// Mitsubishi GX Works2 project: 23_5   PLC: Q03UDV

PROGRAM MAIN
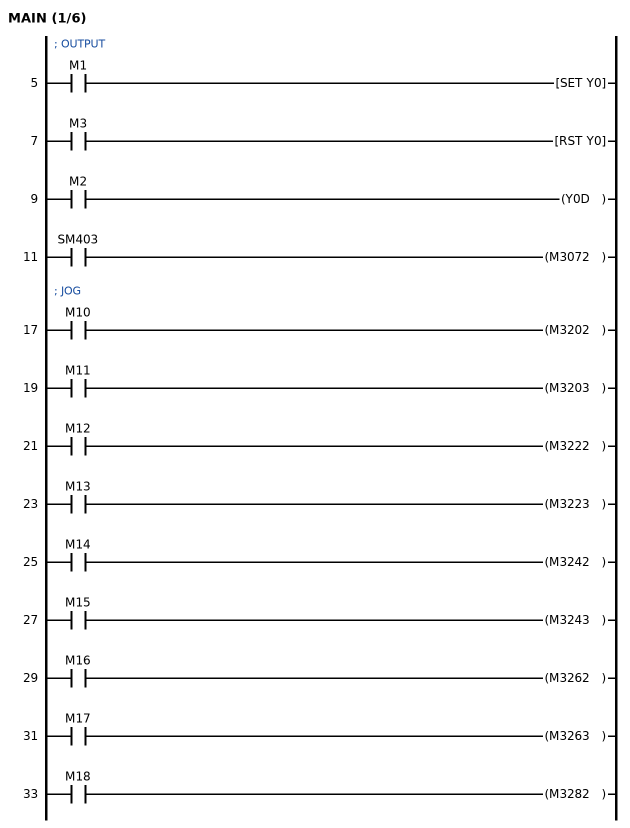
; OUTPUT
5     LD      M1
      SET     Y0
7     LD      M3
      RST     Y0
9     LD      M2
      OUT     Y0D
11    LD      SM403
      OUT     M3072
; JOG
17    LD      M10
      OUT     M3202
19    LD      M11
      OUT     M3203
21    LD      M12
      OUT     M3222
23    LD      M13
      OUT     M3223
25    LD      M14
      OUT     M3242
27    LD      M15
      OUT     M3243
29    LD      M16
      OUT     M3262
31    LD      M17
      OUT     M3263
33    LD      M18
      OUT     M3282
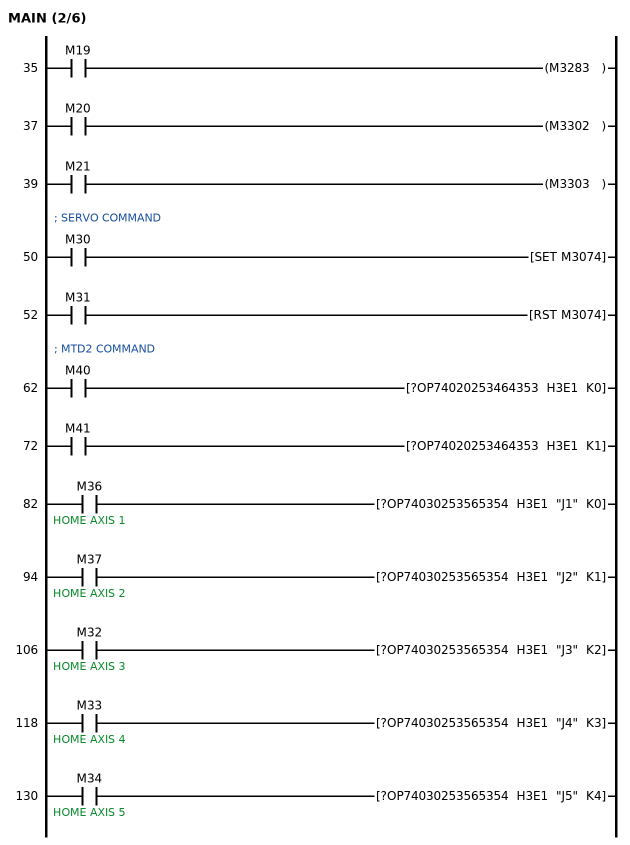
35    LD      M19
      OUT     M3283
37    LD      M20
      OUT     M3302
39    LD      M21
      OUT     M3303
; SERVO COMMAND
50    LD      M30
      SET     M3074
52    LD      M31
      RST     M3074
; MTD2 COMMAND
62    LD      M40
      ?OP74020253464353 H3E1 K0
72    LD      M41
      ?OP74020253464353 H3E1 K1
82    LD      M36  ; HOME AXIS 1
      ?OP74030253565354 H3E1 "J1" K0
94    LD      M37  ; HOME AXIS 2
      ?OP74030253565354 H3E1 "J2" K1
106   LD      M32  ; HOME AXIS 3
      ?OP74030253565354 H3E1 "J3" K2
118   LD      M33  ; HOME AXIS 4
      ?OP74030253565354 H3E1 "J4" K3
130   LD      M34  ; HOME AXIS 5
      ?OP74030253565354 H3E1 "J5" K4
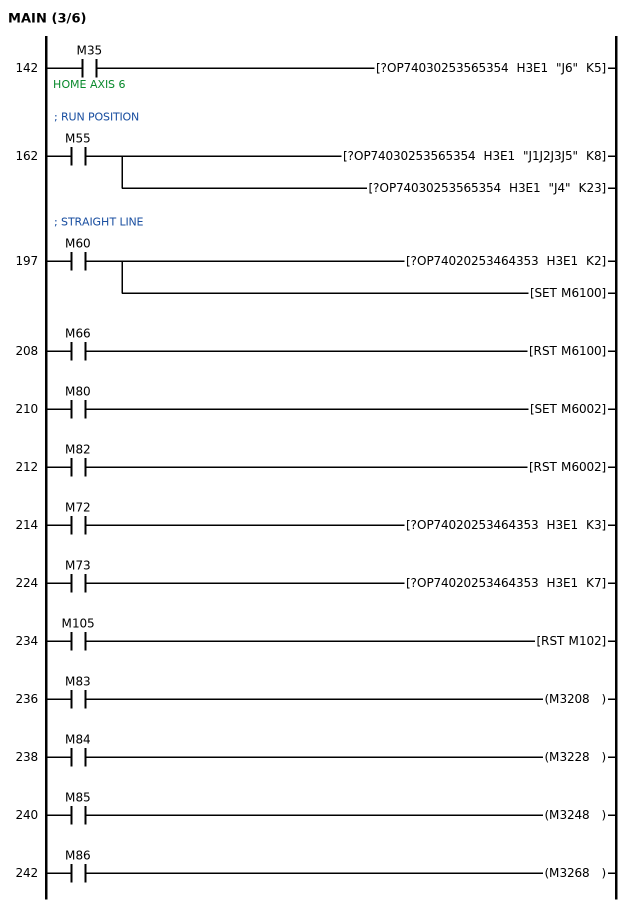
142   LD      M35  ; HOME AXIS 6
      ?OP74030253565354 H3E1 "J6" K5
; RUN POSITION
162   LD      M55
      ?OP74030253565354 H3E1 "J1J2J3J5" K8
      ?OP74030253565354 H3E1 "J4" K23
; STRAIGHT LINE
197   LD      M60
      ?OP74020253464353 H3E1 K2
      SET     M6100
208   LD      M66
      RST     M6100
210   LD      M80
      SET     M6002
212   LD      M82
      RST     M6002
214   LD      M72
      ?OP74020253464353 H3E1 K3
224   LD      M73
      ?OP74020253464353 H3E1 K7
234   LD      M105
      RST     M102
236   LD      M83
      OUT     M3208
238   LD      M84
      OUT     M3228
240   LD      M85
      OUT     M3248
242   LD      M86
      OUT     M3268
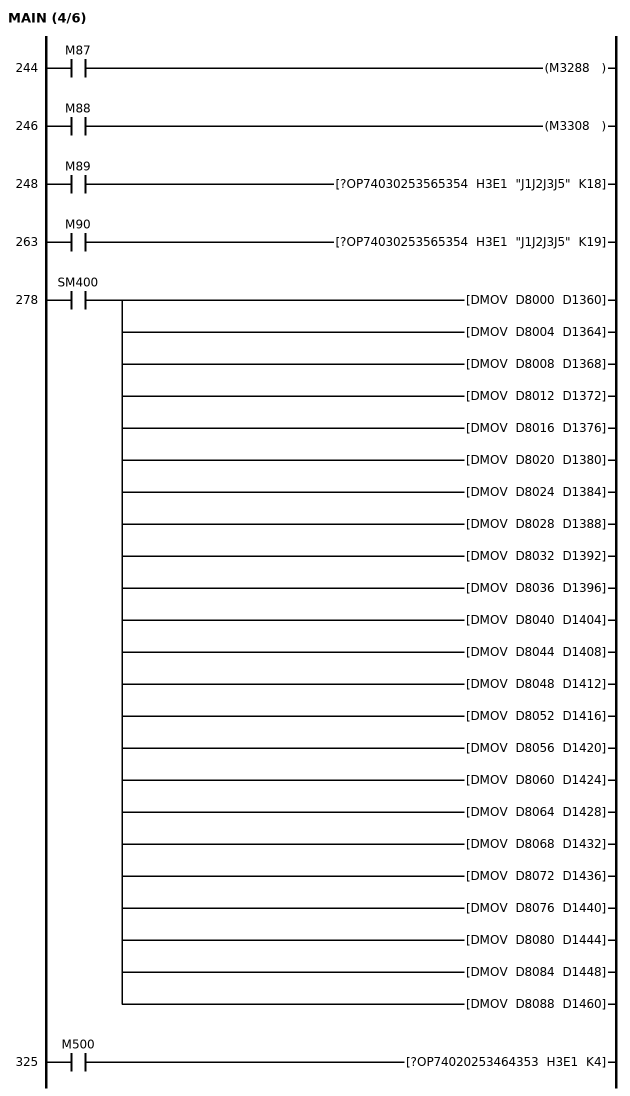
244   LD      M87
      OUT     M3288
246   LD      M88
      OUT     M3308
248   LD      M89
      ?OP74030253565354 H3E1 "J1J2J3J5" K18
263   LD      M90
      ?OP74030253565354 H3E1 "J1J2J3J5" K19
278   LD      SM400
      DMOV    D8000 D1360
      DMOV    D8004 D1364
      DMOV    D8008 D1368
      DMOV    D8012 D1372
      DMOV    D8016 D1376
      DMOV    D8020 D1380
      DMOV    D8024 D1384
      DMOV    D8028 D1388
      DMOV    D8032 D1392
      DMOV    D8036 D1396
      DMOV    D8040 D1404
      DMOV    D8044 D1408
      DMOV    D8048 D1412
      DMOV    D8052 D1416
      DMOV    D8056 D1420
      DMOV    D8060 D1424
      DMOV    D8064 D1428
      DMOV    D8068 D1432
      DMOV    D8072 D1436
      DMOV    D8076 D1440
      DMOV    D8080 D1444
      DMOV    D8084 D1448
      DMOV    D8088 D1460
325   LD      M500
      ?OP74020253464353 H3E1 K4
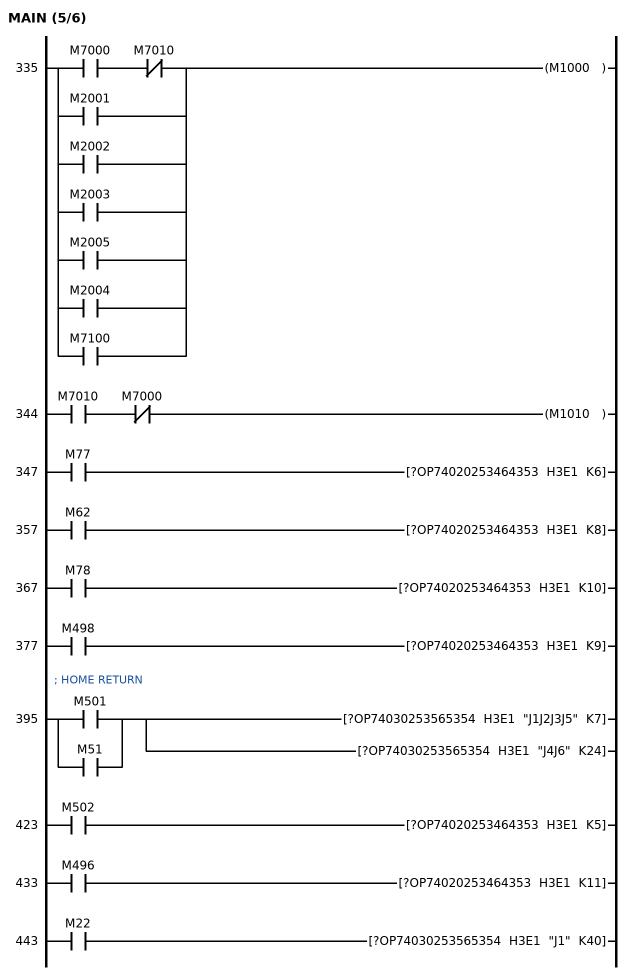
335   LD      M7000
      ANI     M7010
      OR      M2001
      OR      M2002
      OR      M2003
      OR      M2005
      OR      M2004
      OR      M7100
      OUT     M1000
344   LD      M7010
      ANI     M7000
      OUT     M1010
347   LD      M77
      ?OP74020253464353 H3E1 K6
357   LD      M62
      ?OP74020253464353 H3E1 K8
367   LD      M78
      ?OP74020253464353 H3E1 K10
377   LD      M498
      ?OP74020253464353 H3E1 K9
; HOME RETURN
395   LD      M501
      OR      M51
      ?OP74030253565354 H3E1 "J1J2J3J5" K7
      ?OP74030253565354 H3E1 "J4J6" K24
423   LD      M502
      ?OP74020253464353 H3E1 K5
433   LD      M496
      ?OP74020253464353 H3E1 K11
443   LD      M22
      ?OP74030253565354 H3E1 "J1" K40
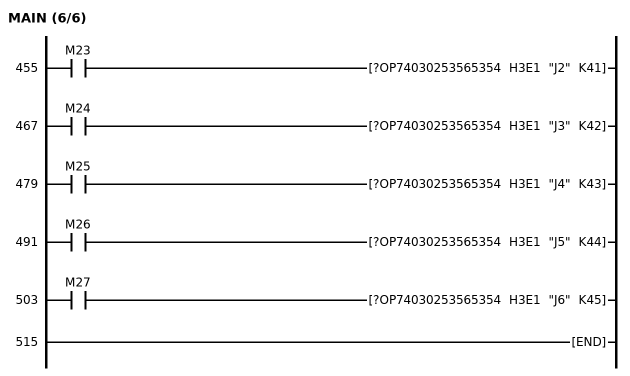
455   LD      M23
      ?OP74030253565354 H3E1 "J2" K41
467   LD      M24
      ?OP74030253565354 H3E1 "J3" K42
479   LD      M25
      ?OP74030253565354 H3E1 "J4" K43
491   LD      M26
      ?OP74030253565354 H3E1 "J5" K44
503   LD      M27
      ?OP74030253565354 H3E1 "J6" K45
515   END
END_PROGRAM
